FUNCTION_BLOCK CmdFeed (* CAT Function Block Type *)
  (* Standard: 61499-2 *)
  (* Version 0.0, 6/7/2026, Schneider Electric, template *)
  PACKAGE SE.Nereda;
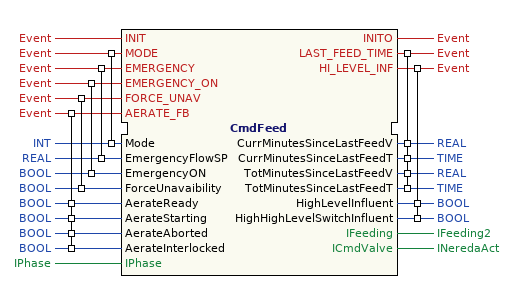
  EVENT_INPUT
    INIT;
    MODE WITH Mode;
    EMERGENCY WITH EmergencyFlowSP;
    EMERGENCY_ON WITH EmergencyON;
    FORCE_UNAV WITH ForceUnavaibility;
    AERATE_FB WITH AerateStarting, AerateAborted, AerateInterlocked, AerateReady;
  END_EVENT
  EVENT_OUTPUT
    INITO;
    LAST_FEED_TIME WITH CurrMinutesSinceLastFeedV, CurrMinutesSinceLastFeedT, TotMinutesSinceLastFeedV, TotMinutesSinceLastFeedT;
    HI_LEVEL_INF WITH HighLevelInfluent, HighHighLevelSwitchInfluent; (* Request from Socket *)
  END_EVENT
  VAR_INPUT
    Mode : INT;
    EmergencyFlowSP : REAL;
    EmergencyON : BOOL;
    ForceUnavaibility : BOOL;
    AerateReady : BOOL;
    AerateStarting : BOOL;
    AerateAborted : BOOL;
    AerateInterlocked : BOOL;
  END_VAR
  VAR_OUTPUT
    CurrMinutesSinceLastFeedV : REAL;
    CurrMinutesSinceLastFeedT : TIME; (* Output event qualifier *)
    TotMinutesSinceLastFeedV : REAL;
    TotMinutesSinceLastFeedT : TIME; (* Output event qualifier *)
    HighLevelInfluent : BOOL; (* Request Data from Socket *)
    HighHighLevelSwitchInfluent : BOOL;
  END_VAR
  SOCKETS
    IPhase : IPhase;
  END_SOCKETS
  PLUGS
    IFeeding : IFeeding2;
  END_PLUGS
  PLUGS
    ICmdValve : INeredaAct;
  END_PLUGS
  (* 01 - FUNCTIONNAL INPUT INTERFACE *)
  (* 00 - INITIALIZATION *)
  (* 05 - LOGIC *)
  (* 06 - HMI INTERFACE *)
  (* 03 - FIELD INTERFACE *)
  (* 02 - FUNCTIONNAL OUTPUT INTERFACE *)
  (* Command Logic *)
  (* Capacity Setpoint *)
  (* Minute Since Last Feed *)
  (* Reset Feed Pump *)
  FBS
    CommandLogic : CmdValvePump; {SET_ATTRIBUTE(Configuration.Component.HideUnusedPorts, )}
    IThis : CmdFeed_HMI(QI := TRUE);
    FeedFlowSpParameterSelector : ParametersSelector;
    TotRunningDurationCalc : devMntCalc(TBaseOperationDuration := T#1s, TBaseElapsedDuration := T#1d); {SET_ATTRIBUTE(Configuration.Component.HideUnusedPorts, )}
    MinutesSinceLastFeed : MinutesSinceLastFeedBasic(pin_2DC2367CDA2D6F18 := 2, pin_0A4BDC38F39F9D58 := TRUE);
    ResetPump : Reset;
    CurrTotDurT : UDINT2TIME_2;
    CurrTotDurV : UDINT2REAL_2;
    CurrRunningDurationCalc : devMntCalc(TBaseOperationDuration := T#1s, TBaseElapsedDuration := T#1d); {SET_ATTRIBUTE(Configuration.Component.HideUnusedPorts, )}
    ResetPulse1 : E_DELAY(DT := T#500ms);
    Tot_s_TO_min : DIVIDE(pin_02E479D09E2C7EA2 := 60);
    Curr_s_TO_min : DIVIDE(pin_02E479D09E2C7EA2 := 60);
    Avaibility : DS_SELECTX_1579ED5B8ACDFC94C; {SET_ATTRIBUTE(Configuration.GenericFBType.InterfaceParams, Runtime.Standard#CNTX:=3;CNTY:=1;DI${CNTX,_,CNTY$}:BOOL)}
    MinutesSinceStartFeed : MinutesSinceLastFeedBasic(pin_2DC2367CDA2D6F18 := 2, pin_0A4BDC38F39F9D58 := FALSE);
    ResetPulse2 : E_DELAY(DT := T#500ms);
    FeedPhase : StartingAborted;
    FeedAerate : StartingAborted;
  END_FBS
  EVENT_CONNECTIONS
    CurrRunningDurationCalc.INITO TO INITO;
    IPhase.Interlocked_CNF TO CommandLogic.CD5317508FB2D68D;
    CommandLogic.20B2DC21F1EA6472 TO IPhase.REQ_Start_Ready;
    CommandLogic.998FBCC53B4D4DC2 TO IPhase.REQ_Stop_Ready;
    CommandLogic.33BFDEBF33D6AC6C TO IPhase.REQ_Abort_Ready;
    MODE TO FeedFlowSpParameterSelector.MODE;
    EMERGENCY TO FeedFlowSpParameterSelector.3B878B7E006C38E4;
    CommandLogic.DB75C281DC5EE23E TO TotRunningDurationCalc.INIT;
    CommandLogic.223351CC605B0EE8 TO IFeeding.74BA0DB8212F2576;
    IFeeding.70EEE9F2AA8AC204 TO CommandLogic.D1EFDB7980E1B3A3;
    IFeeding.70EEE9F2AA8AC204 TO CommandLogic.DADA01CC018E5E78;
    IPhase.Interlocked_CNF TO MinutesSinceLastFeed.D1A4D4DD9A455998;
    IFeeding.03923062E780DBFC TO CommandLogic.D1EFDB7980E1B3A3;
    FeedFlowSpParameterSelector.CNF TO IFeeding.8D6216DA6F1D1AB3;
    INIT TO IThis.C4758748B8B7D3EA;
    CommandLogic.DB75C281DC5EE23E TO IThis.E235583F49B9570B;
    IThis.9FEA1874A72DD629 TO CommandLogic.30F2473D00ED287D;
    IThis.851B32D559A6AA3F TO FeedFlowSpParameterSelector.REQ_NEREDA_VAL;
    IThis.59FB590F9F8A710E TO FeedFlowSpParameterSelector.REQ_MAN_VAL;
    IPhase.Interlocked_CNF TO IFeeding.64A31C18B824409C;
    ResetPump.FEED613FBC3E415D TO IFeeding.9C2DC160D0649F17;
    IPhase.Interlocked_CNF TO ResetPump.BAAD7D98C6D42F1E;
    CurrTotDurV.6FC99A5BD1C38561 TO CurrTotDurT.9954577AA24F9DD6;
    Curr_s_TO_min.6D05A744943B688E TO LAST_FEED_TIME;
    TotRunningDurationCalc.INITO TO CurrRunningDurationCalc.INIT;
    TotRunningDurationCalc.CNF_OPD TO CurrTotDurV.DD5870AA881150BB;
    CurrRunningDurationCalc.CNF_OPD TO CurrTotDurV.DD5870AA881150BB;
    CurrTotDurT.79B40746AB555956 TO Tot_s_TO_min.0FDF8A587C3CA146;
    MinutesSinceLastFeed.9EBF6DD97932C10B TO ResetPulse1.START;
    ResetPulse1.EO TO MinutesSinceLastFeed.C74CA44BB5067CA3;
    MinutesSinceLastFeed.F1D1A71B672AAB1D TO TotRunningDurationCalc.REQ_RESET;
    Tot_s_TO_min.6D05A744943B688E TO Curr_s_TO_min.0FDF8A587C3CA146;
    MinutesSinceLastFeed.75CA504D935A84DB TO TotRunningDurationCalc.REQ_PV;
    MinutesSinceStartFeed.75CA504D935A84DB TO CurrRunningDurationCalc.REQ_PV;
    MinutesSinceStartFeed.F1D1A71B672AAB1D TO CurrRunningDurationCalc.REQ_RESET;
    MinutesSinceStartFeed.9EBF6DD97932C10B TO ResetPulse2.START;
    ResetPulse2.EO TO MinutesSinceStartFeed.C74CA44BB5067CA3;
    CurrRunningDurationCalc.INITO TO MinutesSinceLastFeed.EB976DACF4DE8504;
    CurrRunningDurationCalc.INITO TO MinutesSinceStartFeed.EB976DACF4DE8504;
    IPhase.Interlocked_CNF TO MinutesSinceStartFeed.D1A4D4DD9A455998;
    IPhase.Interlocked_CNF TO FeedPhase.8DB6B3242AA8135A;
    FORCE_UNAV TO Avaibility.REQ1;
    FeedPhase.B3DBBBA4A4378AFC TO Avaibility.REQ2;
    FeedAerate.B3DBBBA4A4378AFC TO Avaibility.REQ3;
    AERATE_FB TO FeedAerate.8DB6B3242AA8135A;
    EMERGENCY_ON TO FeedPhase.8DB6B3242AA8135A;
    EMERGENCY_ON TO FeedAerate.8DB6B3242AA8135A;
    IFeeding.5A11906EF1EE87B0 TO HI_LEVEL_INF;
  END_CONNECTIONS
  DATA_CONNECTIONS
    IPhase.Ready TO CommandLogic.62C98D43CF38EC53;
    IPhase.Starting TO CommandLogic.C52B6A203C1788E2;
    IPhase.Run TO CommandLogic.1275CFBBB3670404;
    IPhase.Stopping TO CommandLogic.050ADE8396657434;
    IPhase.Aborting TO CommandLogic.A678AA8638FC8E4C;
    CommandLogic.FFF2BACA2E6A4B81 TO IPhase.Start_Ready;
    CommandLogic.47BB3439906EF432 TO IPhase.Stop_Ready;
    CommandLogic.80021FFA67DE4B94 TO IPhase.Abort_Ready;
    Mode TO FeedFlowSpParameterSelector.Mode;
    EmergencyFlowSP TO FeedFlowSpParameterSelector.4C6C1BFF70182CBB;
    CommandLogic.882873A6193BACB4 TO IFeeding.9A80F414E2AF6B87;
    IFeeding.15E0B0692568D904 TO CommandLogic.927B12288311A5D9;
    IFeeding.78D0DDD34C9EF9F8 TO CommandLogic.146D10D1F77357CB;
    IFeeding.B41B0731DC9AD731 TO CommandLogic.846AF9B6D3FD4321;
    MinutesSinceLastFeed.AF4A9541A64ED454 TO TotRunningDurationCalc.Pv;
    IPhase.Starting TO MinutesSinceLastFeed.486ACA64D0F65AA0;
    IPhase.Run TO MinutesSinceLastFeed.F7B2FA90A67B4497;
    IPhase.Stopping TO MinutesSinceLastFeed.6E036EF412E3C363;
    FeedFlowSpParameterSelector.ValOut TO IFeeding.D7CF71AAE7A3D95C;
    IThis.48FC57B4BA0AB67A TO FeedFlowSpParameterSelector.NeredaValue;
    IThis.C4072BA96C21EBC0 TO FeedFlowSpParameterSelector.ManValue;
    IPhase.Run TO IFeeding.EAF64D7B7C3D74B7;
    IPhase.Stopping TO IFeeding.7208B850FC6F172F;
    ResetPump.78F11A90675BB1F3 TO IFeeding.48C5E5A256C6457A;
    IPhase.Starting TO ResetPump.6E3779FCEEE15EFE;
    CurrTotDurT.8AC404843F53B283 TO CurrMinutesSinceLastFeedT;
    Curr_s_TO_min.E78A8A65D4120686 TO CurrMinutesSinceLastFeedV;
    CurrRunningDurationCalc.CurrentOperationDuration TO CurrTotDurV.4573FC8F228EB71D;
    TotRunningDurationCalc.TotalOperationDuration TO CurrTotDurV.63EF56506AEB9BC9;
    CurrRunningDurationCalc.CurrentOperationDuration TO CurrTotDurT.158B8AA7B31D2617;
    TotRunningDurationCalc.TotalOperationDuration TO CurrTotDurT.E55D6D2AC87EFFD0;
    Tot_s_TO_min.E78A8A65D4120686 TO TotMinutesSinceLastFeedV;
    CurrTotDurT.4CB3A5FE1D5BD476 TO TotMinutesSinceLastFeedT;
    CurrTotDurV.5DAA0892996D1670 TO Tot_s_TO_min.8EF5C40F2FEA5451;
    CurrTotDurV.A6DEF5F9C27C1848 TO Curr_s_TO_min.8EF5C40F2FEA5451;
    MinutesSinceLastFeed.6A2647797C19ACFF TO TotRunningDurationCalc.ResetOperationDuration;
    MinutesSinceStartFeed.AF4A9541A64ED454 TO CurrRunningDurationCalc.Pv;
    MinutesSinceStartFeed.6A2647797C19ACFF TO CurrRunningDurationCalc.ResetOperationDuration;
    IPhase.Starting TO MinutesSinceStartFeed.486ACA64D0F65AA0;
    IPhase.Run TO MinutesSinceStartFeed.F7B2FA90A67B4497;
    IPhase.Stopping TO MinutesSinceStartFeed.6E036EF412E3C363;
    IPhase.Ready TO FeedPhase.80095D5FE6A4D3E6;
    IPhase.Starting TO FeedPhase.F3E225F6D813FFA6;
    IPhase.Aborted TO FeedPhase.010B04C597ED11DE;
    ForceUnavaibility TO Avaibility.DI1_1;
    IPhase.Interlocked TO FeedPhase.AAC416DA457A1946;
    FeedPhase.3CFCAA7555820094 TO Avaibility.DI2_1;
    FeedAerate.3CFCAA7555820094 TO Avaibility.DI3_1;
    AerateReady TO FeedAerate.80095D5FE6A4D3E6;
    AerateStarting TO FeedAerate.F3E225F6D813FFA6;
    AerateAborted TO FeedAerate.010B04C597ED11DE;
    AerateInterlocked TO FeedAerate.AAC416DA457A1946;
    EmergencyON TO FeedPhase.619E81F440951874;
    EmergencyON TO FeedAerate.619E81F440951874;
    IFeeding.2B9DC646C4F67E84 TO HighLevelInfluent;
  END_CONNECTIONS
  ADAPTER_CONNECTIONS
    CommandLogic.1DFC3C79C26C4936 TO ICmdValve;
  END_CONNECTIONS
END_FUNCTION_BLOCK
